// Mitsubishi GX Works2 project: BookEX6_24 Conversion   PLC: Q13UDV

// global labels: Global
VAR_GLOBAL
  bVar0 AT M5000 : BOOL;
  abArray0 AT M5010 : ARRAY [0..49] OF BOOL;
  sStr0 AT D5000 : STRING[199];
  sStr1 AT D5100 : STRING[199];
  sStr2 AT D5200 : STRING[199];
  sStr3 AT D5300 : STRING[199];
  sStr4 AT D5400 : STRING[199];
  sStr5 AT D5500 : STRING[199];
  sStr6 AT D5600 : STRING[199];
  sStr7 AT D5700 : STRING[199];
  sStr8 AT D5800 : STRING[199];
  sStr9 AT D5900 : STRING[199];
  iVar0 AT D4500 : INT;
  iVar1 AT D4501 : INT;
  iVar2 AT D4502 : INT;
  iVar3 AT D4503 : INT;
  iVar4 AT D4504 : INT;
  iVar5 AT D4505 : INT;
  iVar6 AT D4506 : INT;
  iVar7 AT D4507 : INT;
  iVar8 AT D4508 : INT;
  iVar9 AT D4509 : INT;
  dVar0 AT D4510 : DINT;
  dVar1 AT D4512 : DINT;
  dVar2 AT D4514 : DINT;
  dVar3 AT D4516 : DINT;
  dVar4 AT D4518 : DINT;
  dVar5 AT D4520 : DINT;
  dVar6 AT D4522 : DINT;
  dVar7 AT D4524 : DINT;
  dVar8 AT D4526 : DINT;
  dVar9 AT D4528 : DINT;
  wVar0 AT D4530 : WORD;
  wVar1 AT D4531 : WORD;
  wVar2 AT D4532 : WORD;
  wVar3 AT D4533 : WORD;
  wVar4 AT D4534 : WORD;
  wVar5 AT D4535 : WORD;
  wVar6 AT D4536 : WORD;
  wVar7 AT D4537 : WORD;
  wVar8 AT D4538 : WORD;
  wVar9 AT D4539 : WORD;
  dwVar0 AT D4540 : DWORD;
  dwVar1 AT D4542 : DWORD;
  dwVar2 AT D4544 : DWORD;
  dwVar3 AT D4546 : DWORD;
  dwVar4 AT D4548 : DWORD;
  dwVar5 AT D4550 : DWORD;
  dwVar6 AT D4552 : DWORD;
  dwVar7 AT D4554 : DWORD;
  dwVar8 AT D4556 : DWORD;
  dwVar9 AT D4558 : DWORD;
  fsVar0 AT D4560 : REAL;
  fsVar1 AT D4562 : REAL;
  fsVar2 AT D4564 : REAL;
  fsVar3 AT D4566 : REAL;
  fsVar4 AT D4568 : REAL;
  fsVar5 AT D4570 : REAL;
  fsVar6 AT D4572 : REAL;
  fsVar7 AT D4574 : REAL;
  fsVar8 AT D4576 : REAL;
  fsVar9 AT D4578 : REAL;
  fdVar0 AT D4580 : LREAL;
  tTime0 AT D4620 : TIME;
  tTime1 AT D4622 : TIME;
  tTime2 AT D4624 : TIME;
  tTime3 AT D4626 : TIME;
  tTime4 AT D4628 : TIME;
  tTime5 AT D4630 : TIME;
  tTime6 AT D4632 : TIME;
  tTime7 AT D4634 : TIME;
  tTime8 AT D4636 : TIME;
  tTime9 AT D4638 : TIME;
  tTime10 AT D4640 : TIME;
  bVar1 AT M5001 : BOOL;
  bVar2 AT M5002 : BOOL;
  bVar3 AT M5003 : BOOL;
  bVar4 AT M5004 : BOOL;
  bVar5 AT M5005 : BOOL;
  bVar6 AT M5006 : BOOL;
  bVar7 AT M5007 : BOOL;
  bVar8 AT M5008 : BOOL;
  bVar9 AT M5009 : BOOL;
  abArray1 AT M5060 : ARRAY [0..49] OF BOOL;
  abArray2 AT M5110 : ARRAY [0..49] OF BOOL;
  abArray3 AT M5160 : ARRAY [0..49] OF BOOL;
  abArray4 AT M5210 : ARRAY [0..49] OF BOOL;
  abArray5 AT M5260 : ARRAY [0..49] OF BOOL;
  abArray6 AT M5310 : ARRAY [0..49] OF BOOL;
  abArray7 AT M5360 : ARRAY [0..49] OF BOOL;
  abArray8 AT M5410 : ARRAY [0..49] OF BOOL;
  abArray9 AT M5460 : ARRAY [0..49] OF BOOL;
  fdVar1 AT D4584 : LREAL;
  fdVar2 AT D4588 : LREAL;
  fdVar3 AT D4592 : LREAL;
  fdVar4 AT D4596 : LREAL;
  fdVar5 AT D4600 : LREAL;
  fdVar6 AT D4604 : LREAL;
  fdVar7 AT D4608 : LREAL;
  fdVar8 AT D4612 : LREAL;
  fdVar9 AT D4616 : LREAL;
  afsPen0 AT D2000 : ARRAY [0..499] OF REAL;
  afsPen1 AT D3000 : ARRAY [0..499] OF REAL;
END_VAR
// user libraries (not included): HMI

FUNCTION GRY24
VAR_INPUT
  dw_IN : DWORD;
END_VAR
VAR
  dwTmp : DWORD;
  ix : INT;
  dwRes : DWORD;
  bTmp : BOOL;
END_VAR
;
dwTmp := dw_IN;
DROL(TRUE, 8, dwTmp);
dwRes := 0;
bTmp := FALSE;
FOR ix := 0 TO 23 DO 
	DROL(TRUE, 1, dwRes);
	DROL(TRUE, 1, dwTmp);
	bTmp := SM700 XOR bTmp;
	IF bTmp THEN
		dwRes := dwRes OR 1;
	END_IF;
END_FOR;
GRY24 := dwRes;
END_FUNCTION

PROGRAM ExBCD
VAR
  HMI20_1 : HMI20;
END_VAR
(* structured ladder/FBD written out as ST: instructions are called as NAME(EN, inputs, outputs); _pN, _eN, _tN stand for wires *)
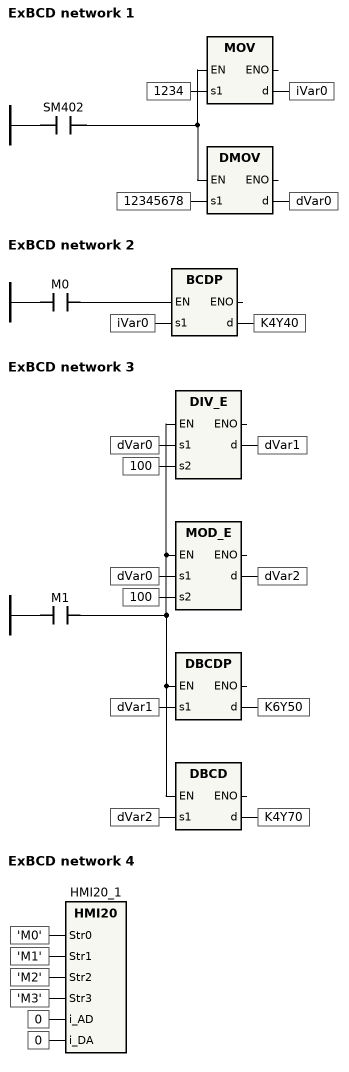
(* network 1 *)
MOV(SM402, 1234, iVar0);
DMOV(SM402, 12345678, dVar0);
(* network 2 *)
BCDP(M0, iVar0, K4Y40);
(* network 3 *)
DIV_E(M1, dVar0, 100, dVar1);
MOD_E(M1, dVar0, 100, dVar2);
DBCDP(M1, dVar1, K6Y50);
DBCD(M1, dVar2, K4Y70);
(* network 4 *)
HMI20_1(Str0 := 'M0', Str1 := 'M1', Str2 := 'M2', Str3 := 'M3', i_AD := 0, i_DA := 0);
END_PROGRAM

PROGRAM ExBIN
VAR
  HMI20_1 : HMI20;
END_VAR
(* structured ladder/FBD written out as ST: instructions are called as NAME(EN, inputs, outputs); _pN, _eN, _tN stand for wires *)
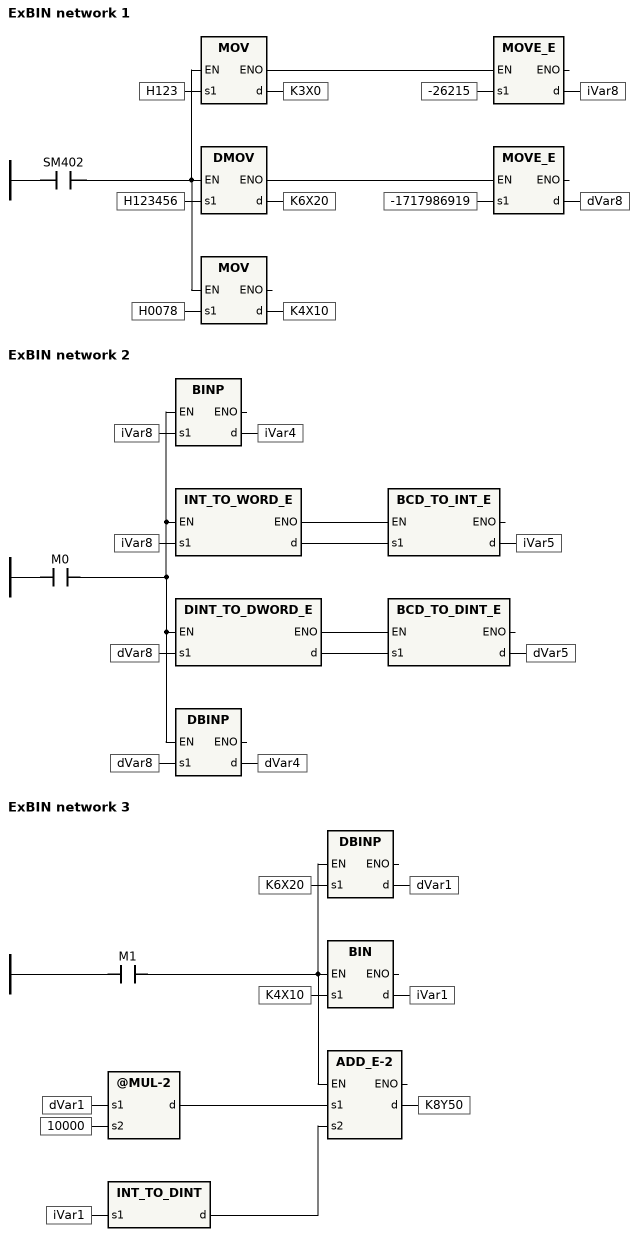
(* network 1 *)
_e1 := MOV(SM402, H123, K3X0);
MOVE_E(_e1, -26215, iVar8);
_e2 := DMOV(SM402, H123456, K6X20);
MOVE_E(_e2, -1717986919, dVar8);
MOV(SM402, H0078, K4X10);
(* network 2 *)
BINP(M0, iVar8, iVar4);
_e2 := INT_TO_WORD_E(M0, iVar8, _t1);
BCD_TO_INT_E(_e2, _t1, iVar5);
DBINP(M0, dVar8, dVar4);
_e4 := DINT_TO_DWORD_E(M0, dVar8, _t3);
BCD_TO_DINT_E(_e4, _t3, dVar5);
(* network 3 *)
DBINP(M1, K6X20, dVar1);
BIN(M1, K4X10, iVar1);
ADD_E(M1, @MUL-2(dVar1, 10000), INT_TO_DINT(iVar1), K8Y50);
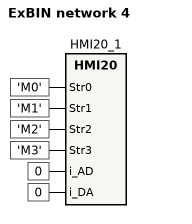
(* network 4 *)
HMI20_1(Str0 := 'M0', Str1 := 'M1', Str2 := 'M2', Str3 := 'M3', i_AD := 0, i_DA := 0);
END_PROGRAM

PROGRAM ExBKBCD
VAR
  Mov4INT_1 : Mov4INT;
  Mov4INT_2 : Mov4INT;
END_VAR
(* structured ladder/FBD written out as ST: instructions are called as NAME(EN, inputs, outputs); _pN, _eN, _tN stand for wires *)
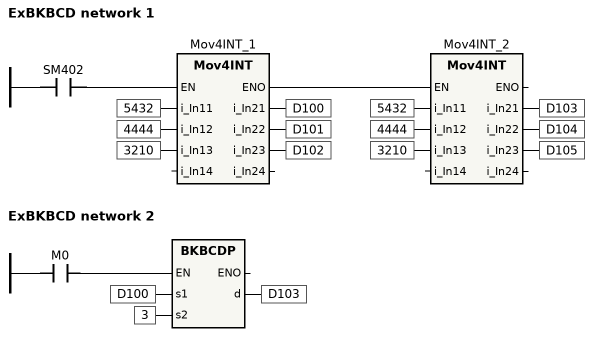
(* network 1 *)
Mov4INT_1(EN := SM402, i_In11 := 5432, i_In12 := 4444, i_In13 := 3210, i_In21 => D100, i_In22 => D101, i_In23 => D102);
Mov4INT_2(EN := Mov4INT_1.ENO, i_In11 := 5432, i_In12 := 4444, i_In13 := 3210, i_In21 => D103, i_In22 => D104, i_In23 => D105);
(* network 2 *)
BKBCDP(M0, D100, 3, D103);
END_PROGRAM

PROGRAM ExBKBIN
VAR
  Mov4INT_1 : Mov4INT;
  Mov4INT_2 : Mov4INT;
END_VAR
(* structured ladder/FBD written out as ST: instructions are called as NAME(EN, inputs, outputs); _pN, _eN, _tN stand for wires *)
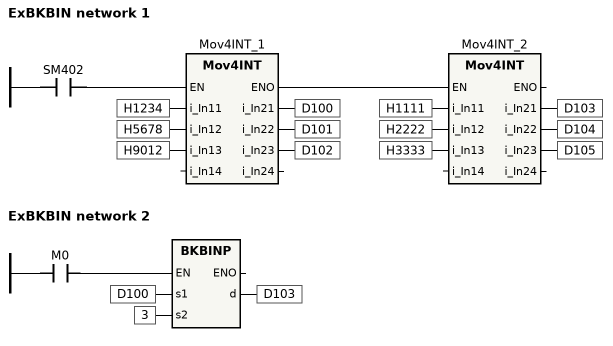
(* network 1 *)
Mov4INT_1(EN := SM402, i_In11 := H1234, i_In12 := H5678, i_In13 := H9012, i_In21 => D100, i_In22 => D101, i_In23 => D102);
Mov4INT_2(EN := Mov4INT_1.ENO, i_In11 := H1111, i_In12 := H2222, i_In13 := H3333, i_In21 => D103, i_In22 => D104, i_In23 => D105);
(* network 2 *)
BKBINP(M0, D100, 3, D103);
END_PROGRAM

PROGRAM ExDBL
(* structured ladder/FBD written out as ST: instructions are called as NAME(EN, inputs, outputs); _pN, _eN, _tN stand for wires *)
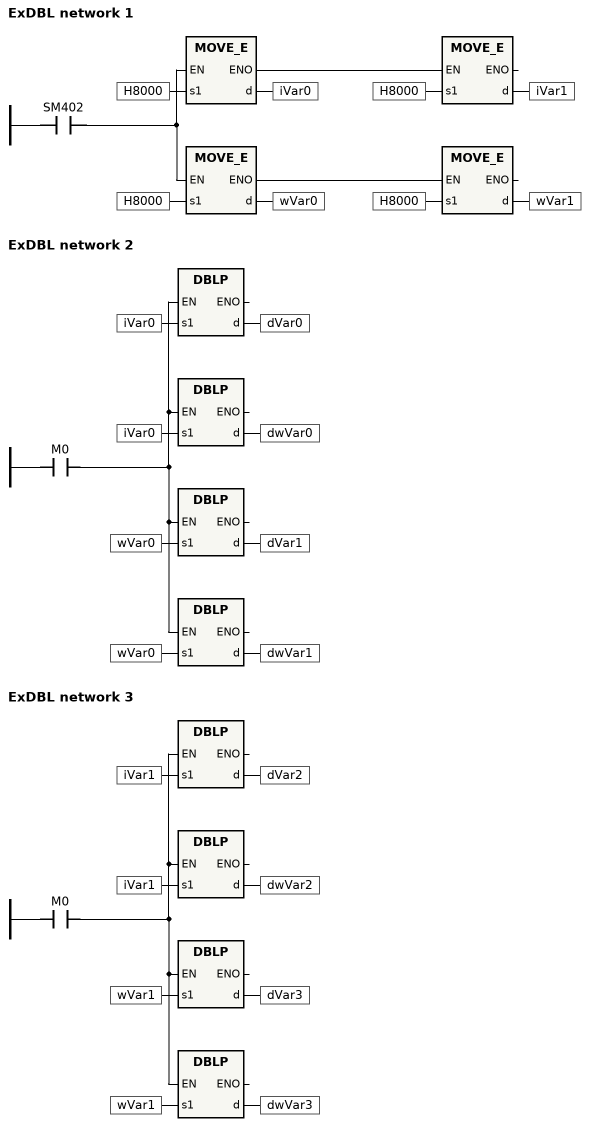
(* network 1 *)
_e1 := MOVE_E(SM402, H8000, iVar0);
MOVE_E(_e1, H8000, iVar1);
_e2 := MOVE_E(SM402, H8000, wVar0);
MOVE_E(_e2, H8000, wVar1);
(* network 2 *)
DBLP(M0, iVar0, dVar0);
DBLP(M0, iVar0, dwVar0);
DBLP(M0, wVar0, dVar1);
DBLP(M0, wVar0, dwVar1);
(* network 3 *)
DBLP(M0, iVar1, dVar2);
DBLP(M0, iVar1, dwVar2);
DBLP(M0, wVar1, dVar3);
DBLP(M0, wVar1, dwVar3);
END_PROGRAM

PROGRAM ExECON
(* structured ladder/FBD written out as ST: instructions are called as NAME(EN, inputs, outputs); _pN, _eN, _tN stand for wires *)
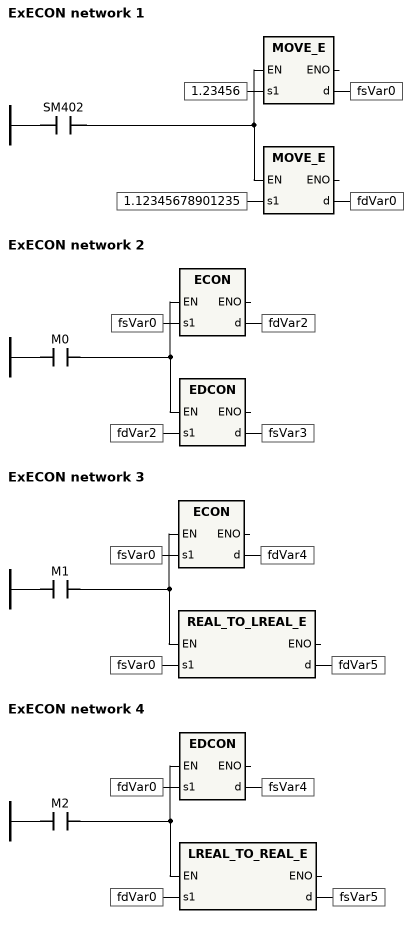
(* network 1 *)
MOVE_E(SM402, 1.23456, fsVar0);
MOVE_E(SM402, 1.12345678901235, fdVar0);
(* network 2 *)
ECON(M0, fsVar0, fdVar2);
EDCON(M0, fdVar2, fsVar3);
(* network 3 *)
ECON(M1, fsVar0, fdVar4);
REAL_TO_LREAL_E(M1, fsVar0, fdVar5);
(* network 4 *)
EDCON(M2, fdVar0, fsVar4);
LREAL_TO_REAL_E(M2, fdVar0, fsVar5);
END_PROGRAM

PROGRAM ExFLT
(* structured ladder/FBD written out as ST: instructions are called as NAME(EN, inputs, outputs); _pN, _eN, _tN stand for wires *)
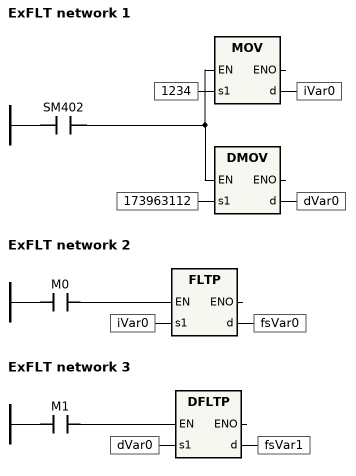
(* network 1 *)
MOV(SM402, 1234, iVar0);
DMOV(SM402, 173963112, dVar0);
(* network 2 *)
FLTP(M0, iVar0, fsVar0);
(* network 3 *)
DFLTP(M1, dVar0, fsVar1);
END_PROGRAM

PROGRAM ExFLTD
(* structured ladder/FBD written out as ST: instructions are called as NAME(EN, inputs, outputs); _pN, _eN, _tN stand for wires *)
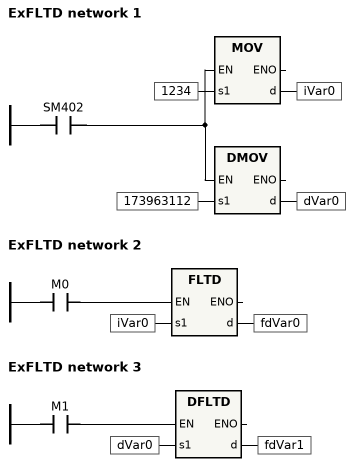
(* network 1 *)
MOV(SM402, 1234, iVar0);
DMOV(SM402, 173963112, dVar0);
(* network 2 *)
FLTD(M0, iVar0, fdVar0);
(* network 3 *)
DFLTD(M1, dVar0, fdVar1);
END_PROGRAM

PROGRAM ExGRY
(* structured ladder/FBD written out as ST: instructions are called as NAME(EN, inputs, outputs); _pN, _eN, _tN stand for wires *)
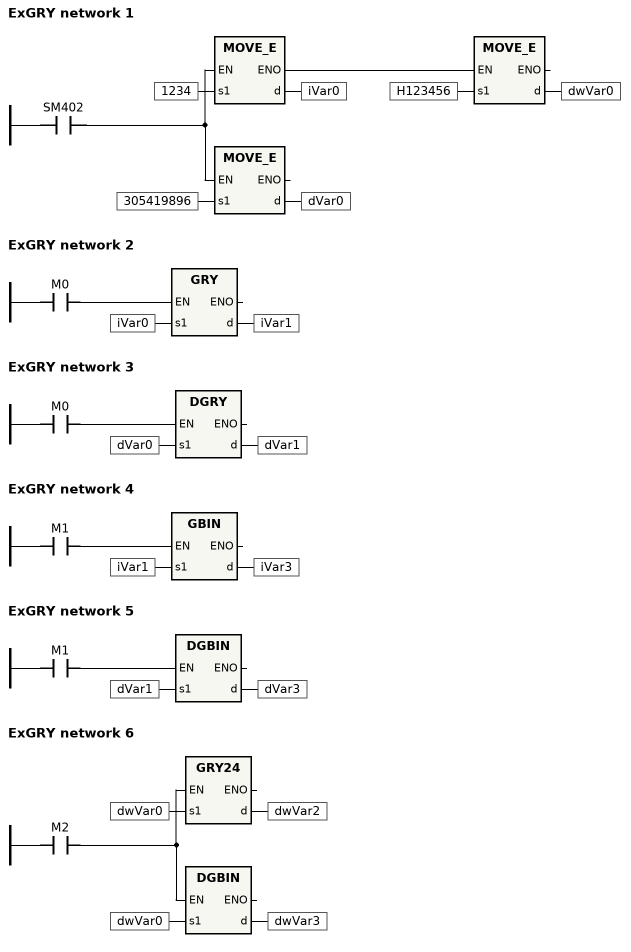
(* network 1 *)
_e1 := MOVE_E(SM402, 1234, iVar0);
MOVE_E(_e1, H123456, dwVar0);
MOVE_E(SM402, 305419896, dVar0);
(* network 2 *)
GRY(M0, iVar0, iVar1);
(* network 3 *)
DGRY(M0, dVar0, dVar1);
(* network 4 *)
GBIN(M1, iVar1, iVar3);
(* network 5 *)
DGBIN(M1, dVar1, dVar3);
(* network 6 *)
GRY24(M2, dwVar0, dwVar2);
DGBIN(M2, dwVar0, dwVar3);
END_PROGRAM

PROGRAM ExINT
(* structured ladder/FBD written out as ST: instructions are called as NAME(EN, inputs, outputs); _pN, _eN, _tN stand for wires *)
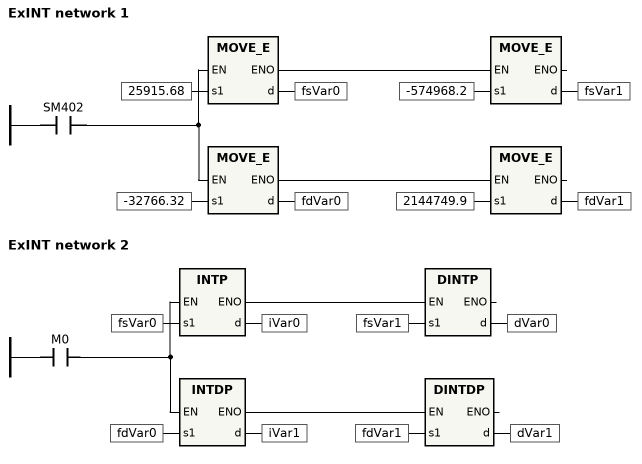
(* network 1 *)
_e1 := MOVE_E(SM402, 25915.68, fsVar0);
MOVE_E(_e1, -574968.2, fsVar1);
_e2 := MOVE_E(SM402, -32766.32, fdVar0);
MOVE_E(_e2, 2144749.9, fdVar1);
(* network 2 *)
_e1 := INTP(M0, fsVar0, iVar0);
DINTP(_e1, fsVar1, dVar0);
_e2 := INTDP(M0, fdVar0, iVar1);
DINTDP(_e2, fdVar1, dVar1);
END_PROGRAM

PROGRAM ExNEG
(* structured ladder/FBD written out as ST: instructions are called as NAME(EN, inputs, outputs); _pN, _eN, _tN stand for wires *)
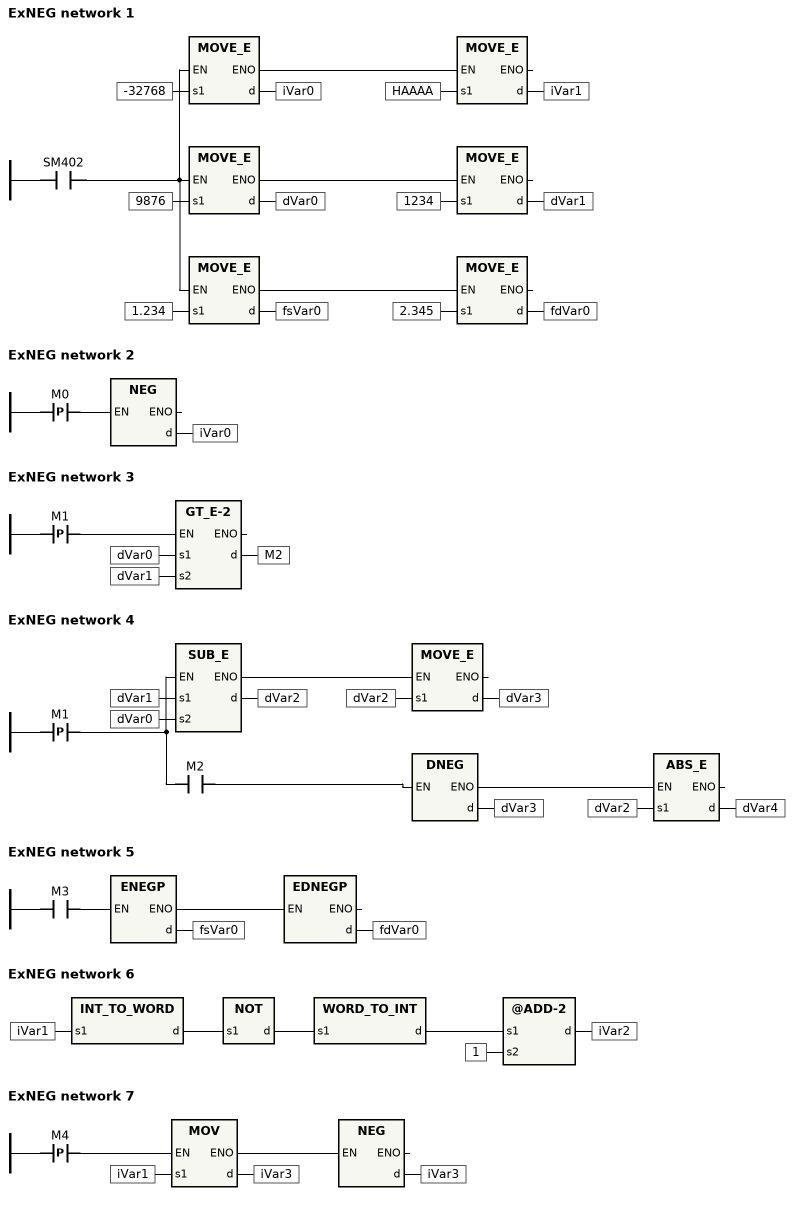
(* network 1 *)
_e1 := MOVE_E(SM402, -32768, iVar0);
MOVE_E(_e1, HAAAA, iVar1);
_e2 := MOVE_E(SM402, 9876, dVar0);
MOVE_E(_e2, 1234, dVar1);
_e3 := MOVE_E(SM402, 1.234, fsVar0);
MOVE_E(_e3, 2.345, fdVar0);
(* network 2 *)
NEG(LDP(TRUE, M0), iVar0);
(* network 3 *)
GT_E(LDP(TRUE, M1), dVar0, dVar1, M2);
(* network 4 *)
_p1 := LDP(TRUE, M1);
_e2 := SUB_E(_p1, dVar1, dVar0, dVar2);
MOVE_E(_e2, dVar2, dVar3);
_e3 := DNEG(_p1 AND M2, dVar3);
ABS_E(_e3, dVar2, dVar4);
(* network 5 *)
_e1 := ENEGP(M3, fsVar0);
EDNEGP(_e1, fdVar0);
(* network 6 *)
iVar2 := @ADD-2(WORD_TO_INT(NOT(INT_TO_WORD(iVar1))), 1);
(* network 7 *)
_e1 := MOV(LDP(TRUE, M4), iVar1, iVar3);
NEG(_e1, iVar3);
END_PROGRAM

PROGRAM ExWORD
(* structured ladder/FBD written out as ST: instructions are called as NAME(EN, inputs, outputs); _pN, _eN, _tN stand for wires *)
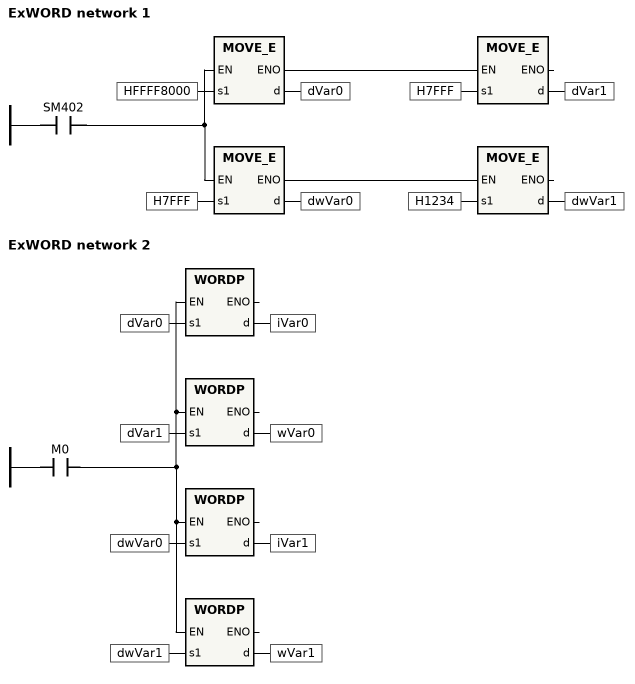
(* network 1 *)
_e1 := MOVE_E(SM402, HFFFF8000, dVar0);
MOVE_E(_e1, H7FFF, dVar1);
_e2 := MOVE_E(SM402, H7FFF, dwVar0);
MOVE_E(_e2, H1234, dwVar1);
(* network 2 *)
WORDP(M0, dVar0, iVar0);
WORDP(M0, dVar1, wVar0);
WORDP(M0, dwVar0, iVar1);
WORDP(M0, dwVar1, wVar1);
END_PROGRAM

PROGRAM ExNEG_ST
;
IF SM402 THEN
	iVar0 := 100;
	dVar0 := 1000;
	fsVar0 := 100.0;
	fdVar0 := 1000.0;
	iVar1 := 500;
	dVar1 := 5000;
	fsVar1 := 500.0;
	fdVar1 := 5000.0;
END_IF;

iVar4 := - iVar0;
dVar4 := - dVar0;
fsVar4 := - fsVar0;
fdVar4 := - fdVar0;

IF LDP(TRUE, M0) THEN
	NEG(TRUE, iVar1);
	DNEG(TRUE, dVar1);
	ENEG(TRUE, fsVar1);
	EDNEG(TRUE, fdVar1);
END_IF;
END_PROGRAM
